TYPE ST_LeakTestRecipe :
STRUCT
	Config : ARRAY[0..GVL_LeakTestConfig.nMaxTestCount] OF ST_RecipeTypeLeakTest;
	Recipe : ARRAY[0..GVL_LeakTestConfig.nMaxTestCount] OF ST_LeakTestStepRecipe;
END_STRUCT
END_TYPE

(* stored: Version 1.1.0.1
   DUT ST_LeakTestRecipe: Id {ea58bc42-04f3-0d40-27a1-f5cea40e895d} *)
